// TwinCAT 3 PLC project Hexapod_Robot_Control_Test
// ProgramVersion: 3.1.4020.4
// libraries:
//   Tc2_MC2, * (Beckhoff Automation GmbH)
//   Tc2_Standard, * (Beckhoff Automation GmbH)
//   Tc2_System, * (Beckhoff Automation GmbH)
//   Tc3_Module, * (Beckhoff Automation GmbH)
//   VisuDialogs, * (System)
// project tree:
//   DUTs/Axis/ Axis.TcPOU (not stored)
//   DUTs/Delay/ Delay.TcPOU (not stored)
//   DUTs/Filter_Current/ E_TcMatSimDataAreaType_1.TcDUT (not stored), FB_Filter_Current_Hexapod_Robot.TcPOU (not stored), FB_TcMatSimObject_1.TcPOU (not stored), ST_Filter_Current_Hexapod_Robot_InitData.TcDUT (not stored), ST_Filter_Current_Hexapod_Robot_Input.TcDUT (not stored), ST_Filter_Current_Hexapod_Robot_Output.TcDUT (not stored), ST_TcMatSimObjectDataAreaInfo_1.TcDUT (not stored)
//   DUTs/Hexapod_Leg/ Hexapod_Leg.TcPOU (not stored)
//   DUTs/Mapping/ Hexapod_Robot_Mapping.TcPOU (not stored)
//   DUTs/Robot_Simulink/ E_TcMatSimDataAreaType.TcDUT, FB_HexMove.TcPOU, FB_TcMatSimObject.TcPOU (not stored), ST_HexMove_InitData.TcDUT (not stored), ST_HexMove_Input.TcDUT (not stored), ST_HexMove_Output.TcDUT, ST_TcMatSimObjectDataAreaInfo.TcDUT
//   / GlobalTextList.TcGTLO, PlcTask.TcTTO, 视图管理器.TcVMO (not stored)
//   POUs/ MAIN.TcPOU
//   VISUs/ Visu_Home.TcVIS (not stored), Visu_SimulinkMove.TcVIS, Visu_Power.TcVIS (not stored), Visu_Reset.TcVIS (not stored), Visu_Stand.TcVIS (not stored)
// real-time tasks:
//   TASK PlcTask: cycle T#1ms, priority 20, ADS port 350
// motion (NC):
//   TASK NC-Task 1 SAF: cycle T#1ms, priority 4, ADS port 501
//   TASK NC-Task 1 SVB: cycle T#1ms, priority 8, ADS port 511
//   AXIS Axis 1 (id 1)
//     Velo: SlowManual=10, FastManual=20
//     OtherSettings: AllowMotionCmdToSlave=true
//     encoder EncType=19
//       EncPara: ScaleFactorNumerator=0.000152590218967, MaxCount=#xffffffff
//     drive DrvType=16
//       DrvPara: MaxCount=#xffffffff
//         TimeComp: TaskDelayCycles=1
//     controller CtrType=1
//       CtrPara: PriorControlFactor=1
//         Observer: BandWidth=20
//   AXIS Axis 2 (id 2)
//     Velo: SlowManual=10, FastManual=20
//     OtherSettings: AllowMotionCmdToSlave=true
//     encoder EncType=19
//       EncPara: ScaleFactorNumerator=0.000152590218967, MaxCount=#xffffffff
//     drive DrvType=16
//       DrvPara: MaxCount=#xffffffff
//         TimeComp: TaskDelayCycles=1
//     controller CtrType=1
//       CtrPara: PriorControlFactor=1
//         Observer: BandWidth=20
//   AXIS Axis 3 (id 3)
//     Velo: SlowManual=10, FastManual=20
//     OtherSettings: AllowMotionCmdToSlave=true
//     encoder EncType=19
//       EncPara: ScaleFactorNumerator=0.000152590218967, MaxCount=#xffffffff
//     drive DrvType=16
//       DrvPara: MaxCount=#xffffffff
//         TimeComp: TaskDelayCycles=1
//     controller CtrType=1
//       CtrPara: PriorControlFactor=1
//         Observer: BandWidth=20
//   AXIS Axis 4 (id 4)
//     Velo: SlowManual=10, FastManual=20
//     OtherSettings: AllowMotionCmdToSlave=true
//     encoder EncType=19
//       EncPara: ScaleFactorNumerator=0.000152590218967, MaxCount=#xffffffff
//     drive DrvType=16
//       DrvPara: MaxCount=#xffffffff
//         TimeComp: TaskDelayCycles=1
//     controller CtrType=1
//       CtrPara: PriorControlFactor=1
//         Observer: BandWidth=20
//   AXIS Axis 5 (id 5)
//     Velo: SlowManual=10, FastManual=20
//     OtherSettings: AllowMotionCmdToSlave=true
//     encoder EncType=19
//       EncPara: ScaleFactorNumerator=0.000152590218967, MaxCount=#xffffffff
//     drive DrvType=16
//       DrvPara: MaxCount=#xffffffff
//         TimeComp: TaskDelayCycles=1
//     controller CtrType=1
//       CtrPara: PriorControlFactor=1
//         Observer: BandWidth=20
//   AXIS Axis 6 (id 6)
//     Velo: SlowManual=10, FastManual=20
//     OtherSettings: AllowMotionCmdToSlave=true
//     encoder EncType=19
//       EncPara: ScaleFactorNumerator=0.000152590218967, MaxCount=#xffffffff
//     drive DrvType=16
//       DrvPara: MaxCount=#xffffffff
//         TimeComp: TaskDelayCycles=1
//     controller CtrType=1
//       CtrPara: PriorControlFactor=1
//         Observer: BandWidth=20
//   AXIS Axis 7 (id 7)
//     Velo: SlowManual=10, FastManual=20
//     OtherSettings: AllowMotionCmdToSlave=true
//     encoder EncType=19
//       EncPara: ScaleFactorNumerator=0.000152590218967, MaxCount=#xffffffff
//     drive DrvType=16
//       DrvPara: MaxCount=#xffffffff
//         TimeComp: TaskDelayCycles=1
//     controller CtrType=1
//       CtrPara: PriorControlFactor=1
//         Observer: BandWidth=20
//   AXIS Axis 8 (id 8)
//     Velo: SlowManual=10, FastManual=20
//     OtherSettings: AllowMotionCmdToSlave=true
//     encoder EncType=19
//       EncPara: ScaleFactorNumerator=0.000152590218967, MaxCount=#xffffffff
//     drive DrvType=16
//       DrvPara: MaxCount=#xffffffff
//         TimeComp: TaskDelayCycles=1
//     controller CtrType=1
//       CtrPara: PriorControlFactor=1
//         Observer: BandWidth=20
//   AXIS Axis 9 (id 9)
//     Velo: SlowManual=10, FastManual=20
//     OtherSettings: AllowMotionCmdToSlave=true
//     encoder EncType=19
//       EncPara: ScaleFactorNumerator=0.000152590218967, MaxCount=#xffffffff
//     drive DrvType=16
//       DrvPara: MaxCount=#xffffffff
//         TimeComp: TaskDelayCycles=1
//     controller CtrType=1
//       CtrPara: PriorControlFactor=1
//         Observer: BandWidth=20
//   AXIS Axis 10 (id 10)
//     Velo: SlowManual=10, FastManual=20
//     OtherSettings: AllowMotionCmdToSlave=true
//     encoder EncType=19
//       EncPara: ScaleFactorNumerator=0.000152590218967, MaxCount=#xffffffff
//     drive DrvType=16
//       DrvPara: MaxCount=#xffffffff
//         TimeComp: TaskDelayCycles=1
//     controller CtrType=1
//       CtrPara: PriorControlFactor=1
//         Observer: BandWidth=20
//   AXIS Axis 11 (id 11)
//     Velo: SlowManual=10, FastManual=20
//     OtherSettings: AllowMotionCmdToSlave=true
//     encoder EncType=19
//       EncPara: ScaleFactorNumerator=0.000152590218967, MaxCount=#xffffffff
//     drive DrvType=16
//       DrvPara: MaxCount=#xffffffff
//         TimeComp: TaskDelayCycles=1
//     controller CtrType=1
//       CtrPara: PriorControlFactor=1
//         Observer: BandWidth=20
//   AXIS Axis 12 (id 12)
//     Velo: SlowManual=10, FastManual=20
//     OtherSettings: AllowMotionCmdToSlave=true
//     encoder EncType=19
//       EncPara: ScaleFactorNumerator=0.000152590218967, MaxCount=#xffffffff
//     drive DrvType=16
//       DrvPara: MaxCount=#xffffffff
//         TimeComp: TaskDelayCycles=1
//     controller CtrType=1
//       CtrPara: PriorControlFactor=1
//         Observer: BandWidth=20
//   AXIS Axis 13 (id 13)
//     Velo: SlowManual=10, FastManual=20
//     OtherSettings: AllowMotionCmdToSlave=true
//     encoder EncType=19
//       EncPara: ScaleFactorNumerator=0.000152590218967, MaxCount=#xffffffff
//     drive DrvType=16
//       DrvPara: MaxCount=#xffffffff
//         TimeComp: TaskDelayCycles=1
//     controller CtrType=1
//       CtrPara: PriorControlFactor=1
//         Observer: BandWidth=20
//   AXIS Axis 14 (id 14)
//     Velo: SlowManual=10, FastManual=20
//     OtherSettings: AllowMotionCmdToSlave=true
//     encoder EncType=19
//       EncPara: ScaleFactorNumerator=0.000152590218967, MaxCount=#xffffffff
//     drive DrvType=16
//       DrvPara: MaxCount=#xffffffff
//         TimeComp: TaskDelayCycles=1
//     controller CtrType=1
//       CtrPara: PriorControlFactor=1
//         Observer: BandWidth=20
//   AXIS Axis 15 (id 15)
//     Velo: SlowManual=10, FastManual=20
//     OtherSettings: AllowMotionCmdToSlave=true
//     encoder EncType=19
//       EncPara: ScaleFactorNumerator=0.000152590218967, MaxCount=#xffffffff
//     drive DrvType=16
//       DrvPara: MaxCount=#xffffffff
//         TimeComp: TaskDelayCycles=1
//     controller CtrType=1
//       CtrPara: PriorControlFactor=1
//         Observer: BandWidth=20
//   AXIS Axis 16 (id 16)
//     Velo: SlowManual=10, FastManual=20
//     OtherSettings: AllowMotionCmdToSlave=true
//     encoder EncType=19
//       EncPara: ScaleFactorNumerator=0.000152590218967, MaxCount=#xffffffff
//     drive DrvType=16
//       DrvPara: MaxCount=#xffffffff
//         TimeComp: TaskDelayCycles=1
//     controller CtrType=1
//       CtrPara: PriorControlFactor=1
//         Observer: BandWidth=20
//   AXIS Axis 17 (id 17)
//     Velo: SlowManual=10, FastManual=20
//     OtherSettings: AllowMotionCmdToSlave=true
//     encoder EncType=19
//       EncPara: ScaleFactorNumerator=0.000152590218967, MaxCount=#xffffffff
//     drive DrvType=16
//       DrvPara: MaxCount=#xffffffff
//         TimeComp: TaskDelayCycles=1
//     controller CtrType=1
//       CtrPara: PriorControlFactor=1
//         Observer: BandWidth=20
//   AXIS Axis 18 (id 18)
//     Velo: SlowManual=10, FastManual=20
//     OtherSettings: AllowMotionCmdToSlave=true
//     encoder EncType=19
//       EncPara: ScaleFactorNumerator=0.000152590218967, MaxCount=#xffffffff
//     drive DrvType=16
//       DrvPara: MaxCount=#xffffffff
//         TimeComp: TaskDelayCycles=1
//     controller CtrType=1
//       CtrPara: PriorControlFactor=1
//         Observer: BandWidth=20
// I/O:
//   DEVICE Device 3 (EtherCAT), AmsNetId 5.41.150.106.4.1
//     Drive 1 (Elmo Drive) [Gold EtherCAT GCON Drive Rev:0x000103F6]
//     Drive 2 (Elmo Drive) [Gold EtherCAT GCON Drive Rev:0x000103F6]
//     Drive 3 (Elmo Drive) [Gold EtherCAT GCON Drive Rev:0x000103F6]
//     Drive 4 (Elmo Drive) [Gold EtherCAT GCON Drive Rev:0x000103F6]
//     Drive 5 (Elmo Drive) [Gold EtherCAT GCON Drive Rev:0x000103F6]
//     Drive 6 (Elmo Drive) [Gold EtherCAT GCON Drive Rev:0x000103F6]
//     Drive 7 (Elmo Drive) [Gold EtherCAT GCON Drive Rev:0x000103F6]
//     Drive 8 (Elmo Drive) [Gold EtherCAT GCON Drive Rev:0x000103F6]
//     Drive 9 (Elmo Drive) [Gold EtherCAT GCON Drive Rev:0x000103F6]
//     Drive 10 (Elmo Drive) [Gold EtherCAT GCON Drive Rev:0x000103F6]
//     Drive 11 (Elmo Drive) [Gold EtherCAT GCON Drive Rev:0x000103F6]
//     Drive 12 (Elmo Drive) [Gold EtherCAT GCON Drive Rev:0x000103F6]
//     Drive 13 (Elmo Drive) [Gold EtherCAT GCON Drive Rev:0x000103F6]
//     Drive 14 (Elmo Drive) [Gold EtherCAT GCON Drive Rev:0x000103F6]
//     Drive 15 (Elmo Drive) [Gold EtherCAT GCON Drive Rev:0x000103F6]
//     Drive 16 (Elmo Drive) [Gold EtherCAT GCON Drive Rev:0x000103F6]
//     Drive 17 (Elmo Drive) [Gold EtherCAT GCON Drive Rev:0x000103F6]
//     Drive 18 (Elmo Drive) [Gold EtherCAT GCON Drive Rev:0x000103F6]
// variable links:
//   NC-Task 1 SAF/Axes/Axis 1 <-> Device 3 (EtherCAT)/Drive 1 (Elmo Drive)
//     Drive/Inputs/In/nDcOutputTime <-> InfoData/DcOutputShift
//     Drive/Inputs/In/nState1 <-> Inputs/Status word
//     Drive/Inputs/In/nState2 <-> Inputs/Status word @bit 8
//     Drive/Inputs/In/nState4 @bit 1 <-> WcState/InputToggle
//     Drive/Inputs/In/nState4 <-> WcState/WcState
//     Drive/Outputs/Out/nCtrl1 <-> Outputs/Control word
//     Drive/Outputs/Out/nCtrl2 <-> Outputs/Control word @bit 8
//     Drive/Outputs/Out/nDataOut1 <-> Outputs/Target Position
//     Enc/Inputs/In/nDataIn1 <-> Inputs/Position actual value
//     Enc/Inputs/In/nDcInputTime <-> InfoData/DcInputShift
//     Enc/Inputs/In/nState4 @bit 1 <-> WcState/InputToggle
//     Enc/Inputs/In/nState4 <-> WcState/WcState
//   NC-Task 1 SAF/Axes/Axis 10 <-> Device 3 (EtherCAT)/Drive 10 (Elmo Drive)
//     Drive/Inputs/In/nDcOutputTime <-> InfoData/DcOutputShift
//     Drive/Inputs/In/nState1 <-> Inputs/Status word
//     Drive/Inputs/In/nState2 <-> Inputs/Status word @bit 8
//     Drive/Inputs/In/nState4 @bit 1 <-> WcState/InputToggle
//     Drive/Inputs/In/nState4 <-> WcState/WcState
//     Drive/Outputs/Out/nCtrl1 <-> Outputs/Control word
//     Drive/Outputs/Out/nCtrl2 <-> Outputs/Control word @bit 8
//     Drive/Outputs/Out/nDataOut1 <-> Outputs/Target Position
//     Enc/Inputs/In/nDataIn1 <-> Inputs/Position actual value
//     Enc/Inputs/In/nDcInputTime <-> InfoData/DcInputShift
//     Enc/Inputs/In/nState4 @bit 1 <-> WcState/InputToggle
//     Enc/Inputs/In/nState4 <-> WcState/WcState
//   NC-Task 1 SAF/Axes/Axis 11 <-> Device 3 (EtherCAT)/Drive 11 (Elmo Drive)
//     Drive/Inputs/In/nDcOutputTime <-> InfoData/DcOutputShift
//     Drive/Inputs/In/nState1 <-> Inputs/Status word
//     Drive/Inputs/In/nState2 <-> Inputs/Status word @bit 8
//     Drive/Inputs/In/nState4 @bit 1 <-> WcState/InputToggle
//     Drive/Inputs/In/nState4 <-> WcState/WcState
//     Drive/Outputs/Out/nCtrl1 <-> Outputs/Control word
//     Drive/Outputs/Out/nCtrl2 <-> Outputs/Control word @bit 8
//     Drive/Outputs/Out/nDataOut1 <-> Outputs/Target Position
//     Enc/Inputs/In/nDataIn1 <-> Inputs/Position actual value
//     Enc/Inputs/In/nDcInputTime <-> InfoData/DcInputShift
//     Enc/Inputs/In/nState4 @bit 1 <-> WcState/InputToggle
//     Enc/Inputs/In/nState4 <-> WcState/WcState
//   NC-Task 1 SAF/Axes/Axis 12 <-> Device 3 (EtherCAT)/Drive 12 (Elmo Drive)
//     Drive/Inputs/In/nDcOutputTime <-> InfoData/DcOutputShift
//     Drive/Inputs/In/nState1 <-> Inputs/Status word
//     Drive/Inputs/In/nState2 <-> Inputs/Status word @bit 8
//     Drive/Inputs/In/nState4 @bit 1 <-> WcState/InputToggle
//     Drive/Inputs/In/nState4 <-> WcState/WcState
//     Drive/Outputs/Out/nCtrl1 <-> Outputs/Control word
//     Drive/Outputs/Out/nCtrl2 <-> Outputs/Control word @bit 8
//     Drive/Outputs/Out/nDataOut1 <-> Outputs/Target Position
//     Enc/Inputs/In/nDataIn1 <-> Inputs/Position actual value
//     Enc/Inputs/In/nDcInputTime <-> InfoData/DcInputShift
//     Enc/Inputs/In/nState4 @bit 1 <-> WcState/InputToggle
//     Enc/Inputs/In/nState4 <-> WcState/WcState
//   NC-Task 1 SAF/Axes/Axis 13 <-> Device 3 (EtherCAT)/Drive 13 (Elmo Drive)
//     Drive/Inputs/In/nDcOutputTime <-> InfoData/DcOutputShift
//     Drive/Inputs/In/nState1 <-> Inputs/Status word
//     Drive/Inputs/In/nState2 <-> Inputs/Status word @bit 8
//     Drive/Inputs/In/nState4 @bit 1 <-> WcState/InputToggle
//     Drive/Inputs/In/nState4 <-> WcState/WcState
//     Drive/Outputs/Out/nCtrl1 <-> Outputs/Control word
//     Drive/Outputs/Out/nCtrl2 <-> Outputs/Control word @bit 8
//     Drive/Outputs/Out/nDataOut1 <-> Outputs/Target Position
//     Enc/Inputs/In/nDataIn1 <-> Inputs/Position actual value
//     Enc/Inputs/In/nDcInputTime <-> InfoData/DcInputShift
//     Enc/Inputs/In/nState4 @bit 1 <-> WcState/InputToggle
//     Enc/Inputs/In/nState4 <-> WcState/WcState
//   NC-Task 1 SAF/Axes/Axis 14 <-> Device 3 (EtherCAT)/Drive 14 (Elmo Drive)
//     Drive/Inputs/In/nDcOutputTime <-> InfoData/DcOutputShift
//     Drive/Inputs/In/nState1 <-> Inputs/Status word
//     Drive/Inputs/In/nState2 <-> Inputs/Status word @bit 8
//     Drive/Inputs/In/nState4 @bit 1 <-> WcState/InputToggle
//     Drive/Inputs/In/nState4 <-> WcState/WcState
//     Drive/Outputs/Out/nCtrl1 <-> Outputs/Control word
//     Drive/Outputs/Out/nCtrl2 <-> Outputs/Control word @bit 8
//     Drive/Outputs/Out/nDataOut1 <-> Outputs/Target Position
//     Enc/Inputs/In/nDataIn1 <-> Inputs/Position actual value
//     Enc/Inputs/In/nDcInputTime <-> InfoData/DcInputShift
//     Enc/Inputs/In/nState4 @bit 1 <-> WcState/InputToggle
//     Enc/Inputs/In/nState4 <-> WcState/WcState
//   NC-Task 1 SAF/Axes/Axis 15 <-> Device 3 (EtherCAT)/Drive 15 (Elmo Drive)
//     Drive/Inputs/In/nDcOutputTime <-> InfoData/DcOutputShift
//     Drive/Inputs/In/nState1 <-> Inputs/Status word
//     Drive/Inputs/In/nState2 <-> Inputs/Status word @bit 8
//     Drive/Inputs/In/nState4 @bit 1 <-> WcState/InputToggle
//     Drive/Inputs/In/nState4 <-> WcState/WcState
//     Drive/Outputs/Out/nCtrl1 <-> Outputs/Control word
//     Drive/Outputs/Out/nCtrl2 <-> Outputs/Control word @bit 8
//     Drive/Outputs/Out/nDataOut1 <-> Outputs/Target Position
//     Enc/Inputs/In/nDataIn1 <-> Inputs/Position actual value
//     Enc/Inputs/In/nDcInputTime <-> InfoData/DcInputShift
//     Enc/Inputs/In/nState4 @bit 1 <-> WcState/InputToggle
//     Enc/Inputs/In/nState4 <-> WcState/WcState
//   NC-Task 1 SAF/Axes/Axis 16 <-> Device 3 (EtherCAT)/Drive 16 (Elmo Drive)
//     Drive/Inputs/In/nDcOutputTime <-> InfoData/DcOutputShift
//     Drive/Inputs/In/nState1 <-> Inputs/Status word
//     Drive/Inputs/In/nState2 <-> Inputs/Status word @bit 8
//     Drive/Inputs/In/nState4 @bit 1 <-> WcState/InputToggle
//     Drive/Inputs/In/nState4 <-> WcState/WcState
//     Drive/Outputs/Out/nCtrl1 <-> Outputs/Control word
//     Drive/Outputs/Out/nCtrl2 <-> Outputs/Control word @bit 8
//     Drive/Outputs/Out/nDataOut1 <-> Outputs/Target Position
//     Enc/Inputs/In/nDataIn1 <-> Inputs/Position actual value
//     Enc/Inputs/In/nDcInputTime <-> InfoData/DcInputShift
//     Enc/Inputs/In/nState4 @bit 1 <-> WcState/InputToggle
//     Enc/Inputs/In/nState4 <-> WcState/WcState
//   NC-Task 1 SAF/Axes/Axis 17 <-> Device 3 (EtherCAT)/Drive 17 (Elmo Drive)
//     Drive/Inputs/In/nDcOutputTime <-> InfoData/DcOutputShift
//     Drive/Inputs/In/nState1 <-> Inputs/Status word
//     Drive/Inputs/In/nState2 <-> Inputs/Status word @bit 8
//     Drive/Inputs/In/nState4 @bit 1 <-> WcState/InputToggle
//     Drive/Inputs/In/nState4 <-> WcState/WcState
//     Drive/Outputs/Out/nCtrl1 <-> Outputs/Control word
//     Drive/Outputs/Out/nCtrl2 <-> Outputs/Control word @bit 8
//     Drive/Outputs/Out/nDataOut1 <-> Outputs/Target Position
//     Enc/Inputs/In/nDataIn1 <-> Inputs/Position actual value
//     Enc/Inputs/In/nDcInputTime <-> InfoData/DcInputShift
//     Enc/Inputs/In/nState4 @bit 1 <-> WcState/InputToggle
//     Enc/Inputs/In/nState4 <-> WcState/WcState
//   NC-Task 1 SAF/Axes/Axis 18 <-> Device 3 (EtherCAT)/Drive 18 (Elmo Drive)
//     Drive/Inputs/In/nDcOutputTime <-> InfoData/DcOutputShift
//     Drive/Inputs/In/nState1 <-> Inputs/Status word
//     Drive/Inputs/In/nState2 <-> Inputs/Status word @bit 8
//     Drive/Inputs/In/nState4 @bit 1 <-> WcState/InputToggle
//     Drive/Inputs/In/nState4 <-> WcState/WcState
//     Drive/Outputs/Out/nCtrl1 <-> Outputs/Control word
//     Drive/Outputs/Out/nCtrl2 <-> Outputs/Control word @bit 8
//     Drive/Outputs/Out/nDataOut1 <-> Outputs/Target Position
//     Enc/Inputs/In/nDataIn1 <-> Inputs/Position actual value
//     Enc/Inputs/In/nDcInputTime <-> InfoData/DcInputShift
//     Enc/Inputs/In/nState4 @bit 1 <-> WcState/InputToggle
//     Enc/Inputs/In/nState4 <-> WcState/WcState
//   NC-Task 1 SAF/Axes/Axis 2 <-> Device 3 (EtherCAT)/Drive 2 (Elmo Drive)
//     Drive/Inputs/In/nDcOutputTime <-> InfoData/DcOutputShift
//     Drive/Inputs/In/nState1 <-> Inputs/Status word
//     Drive/Inputs/In/nState2 <-> Inputs/Status word @bit 8
//     Drive/Inputs/In/nState4 @bit 1 <-> WcState/InputToggle
//     Drive/Inputs/In/nState4 <-> WcState/WcState
//     Drive/Outputs/Out/nCtrl1 <-> Outputs/Control word
//     Drive/Outputs/Out/nCtrl2 <-> Outputs/Control word @bit 8
//     Drive/Outputs/Out/nDataOut1 <-> Outputs/Target Position
//     Enc/Inputs/In/nDataIn1 <-> Inputs/Position actual value
//     Enc/Inputs/In/nDcInputTime <-> InfoData/DcInputShift
//     Enc/Inputs/In/nState4 @bit 1 <-> WcState/InputToggle
//     Enc/Inputs/In/nState4 <-> WcState/WcState
//   NC-Task 1 SAF/Axes/Axis 3 <-> Device 3 (EtherCAT)/Drive 3 (Elmo Drive)
//     Drive/Inputs/In/nDcOutputTime <-> InfoData/DcOutputShift
//     Drive/Inputs/In/nState1 <-> Inputs/Status word
//     Drive/Inputs/In/nState2 <-> Inputs/Status word @bit 8
//     Drive/Inputs/In/nState4 @bit 1 <-> WcState/InputToggle
//     Drive/Inputs/In/nState4 <-> WcState/WcState
//     Drive/Outputs/Out/nCtrl1 <-> Outputs/Control word
//     Drive/Outputs/Out/nCtrl2 <-> Outputs/Control word @bit 8
//     Drive/Outputs/Out/nDataOut1 <-> Outputs/Target Position
//     Enc/Inputs/In/nDataIn1 <-> Inputs/Position actual value
//     Enc/Inputs/In/nDcInputTime <-> InfoData/DcInputShift
//     Enc/Inputs/In/nState4 @bit 1 <-> WcState/InputToggle
//     Enc/Inputs/In/nState4 <-> WcState/WcState
//   NC-Task 1 SAF/Axes/Axis 4 <-> Device 3 (EtherCAT)/Drive 4 (Elmo Drive)
//     Drive/Inputs/In/nDcOutputTime <-> InfoData/DcOutputShift
//     Drive/Inputs/In/nState1 <-> Inputs/Status word
//     Drive/Inputs/In/nState2 <-> Inputs/Status word @bit 8
//     Drive/Inputs/In/nState4 @bit 1 <-> WcState/InputToggle
//     Drive/Inputs/In/nState4 <-> WcState/WcState
//     Drive/Outputs/Out/nCtrl1 <-> Outputs/Control word
//     Drive/Outputs/Out/nCtrl2 <-> Outputs/Control word @bit 8
//     Drive/Outputs/Out/nDataOut1 <-> Outputs/Target Position
//     Enc/Inputs/In/nDataIn1 <-> Inputs/Position actual value
//     Enc/Inputs/In/nDcInputTime <-> InfoData/DcInputShift
//     Enc/Inputs/In/nState4 @bit 1 <-> WcState/InputToggle
//     Enc/Inputs/In/nState4 <-> WcState/WcState
//   NC-Task 1 SAF/Axes/Axis 5 <-> Device 3 (EtherCAT)/Drive 5 (Elmo Drive)
//     Drive/Inputs/In/nDcOutputTime <-> InfoData/DcOutputShift
//     Drive/Inputs/In/nState1 <-> Inputs/Status word
//     Drive/Inputs/In/nState2 <-> Inputs/Status word @bit 8
//     Drive/Inputs/In/nState4 @bit 1 <-> WcState/InputToggle
//     Drive/Inputs/In/nState4 <-> WcState/WcState
//     Drive/Outputs/Out/nCtrl1 <-> Outputs/Control word
//     Drive/Outputs/Out/nCtrl2 <-> Outputs/Control word @bit 8
//     Drive/Outputs/Out/nDataOut1 <-> Outputs/Target Position
//     Enc/Inputs/In/nDataIn1 <-> Inputs/Position actual value
//     Enc/Inputs/In/nDcInputTime <-> InfoData/DcInputShift
//     Enc/Inputs/In/nState4 @bit 1 <-> WcState/InputToggle
//     Enc/Inputs/In/nState4 <-> WcState/WcState
//   NC-Task 1 SAF/Axes/Axis 6 <-> Device 3 (EtherCAT)/Drive 6 (Elmo Drive)
//     Drive/Inputs/In/nDcOutputTime <-> InfoData/DcOutputShift
//     Drive/Inputs/In/nState1 <-> Inputs/Status word
//     Drive/Inputs/In/nState2 <-> Inputs/Status word @bit 8
//     Drive/Inputs/In/nState4 @bit 1 <-> WcState/InputToggle
//     Drive/Inputs/In/nState4 <-> WcState/WcState
//     Drive/Outputs/Out/nCtrl1 <-> Outputs/Control word
//     Drive/Outputs/Out/nCtrl2 <-> Outputs/Control word @bit 8
//     Drive/Outputs/Out/nDataOut1 <-> Outputs/Target Position
//     Enc/Inputs/In/nDataIn1 <-> Inputs/Position actual value
//     Enc/Inputs/In/nDcInputTime <-> InfoData/DcInputShift
//     Enc/Inputs/In/nState4 @bit 1 <-> WcState/InputToggle
//     Enc/Inputs/In/nState4 <-> WcState/WcState
//   NC-Task 1 SAF/Axes/Axis 7 <-> Device 3 (EtherCAT)/Drive 7 (Elmo Drive)
//     Drive/Inputs/In/nDcOutputTime <-> InfoData/DcOutputShift
//     Drive/Inputs/In/nState1 <-> Inputs/Status word
//     Drive/Inputs/In/nState2 <-> Inputs/Status word @bit 8
//     Drive/Inputs/In/nState4 @bit 1 <-> WcState/InputToggle
//     Drive/Inputs/In/nState4 <-> WcState/WcState
//     Drive/Outputs/Out/nCtrl1 <-> Outputs/Control word
//     Drive/Outputs/Out/nCtrl2 <-> Outputs/Control word @bit 8
//     Drive/Outputs/Out/nDataOut1 <-> Outputs/Target Position
//     Enc/Inputs/In/nDataIn1 <-> Inputs/Position actual value
//     Enc/Inputs/In/nDcInputTime <-> InfoData/DcInputShift
//     Enc/Inputs/In/nState4 @bit 1 <-> WcState/InputToggle
//     Enc/Inputs/In/nState4 <-> WcState/WcState
//   NC-Task 1 SAF/Axes/Axis 8 <-> Device 3 (EtherCAT)/Drive 8 (Elmo Drive)
//     Drive/Inputs/In/nDcOutputTime <-> InfoData/DcOutputShift
//     Drive/Inputs/In/nState1 <-> Inputs/Status word
//     Drive/Inputs/In/nState2 <-> Inputs/Status word @bit 8
//     Drive/Inputs/In/nState4 @bit 1 <-> WcState/InputToggle
//     Drive/Inputs/In/nState4 <-> WcState/WcState
//     Drive/Outputs/Out/nCtrl1 <-> Outputs/Control word
//     Drive/Outputs/Out/nCtrl2 <-> Outputs/Control word @bit 8
//     Drive/Outputs/Out/nDataOut1 <-> Outputs/Target Position
//     Enc/Inputs/In/nDataIn1 <-> Inputs/Position actual value
//     Enc/Inputs/In/nDcInputTime <-> InfoData/DcInputShift
//     Enc/Inputs/In/nState4 @bit 1 <-> WcState/InputToggle
//     Enc/Inputs/In/nState4 <-> WcState/WcState
//   NC-Task 1 SAF/Axes/Axis 9 <-> Device 3 (EtherCAT)/Drive 9 (Elmo Drive)
//     Drive/Inputs/In/nDcOutputTime <-> InfoData/DcOutputShift
//     Drive/Inputs/In/nState1 <-> Inputs/Status word
//     Drive/Inputs/In/nState2 <-> Inputs/Status word @bit 8
//     Drive/Inputs/In/nState4 @bit 1 <-> WcState/InputToggle
//     Drive/Inputs/In/nState4 <-> WcState/WcState
//     Drive/Outputs/Out/nCtrl1 <-> Outputs/Control word
//     Drive/Outputs/Out/nCtrl2 <-> Outputs/Control word @bit 8
//     Drive/Outputs/Out/nDataOut1 <-> Outputs/Target Position
//     Enc/Inputs/In/nDataIn1 <-> Inputs/Position actual value
//     Enc/Inputs/In/nDcInputTime <-> InfoData/DcInputShift
//     Enc/Inputs/In/nState4 @bit 1 <-> WcState/InputToggle
//     Enc/Inputs/In/nState4 <-> WcState/WcState
//   Hexapod_Robot_Control_Test/Hexapod_Robot_Control_Test Instance <-> Device 3 (EtherCAT)/Drive 1 (Elmo Drive)
//     PlcTask Inputs/MAIN.Current_Turque_Value[1] <-> Inputs_1/Current actual value
//   Hexapod_Robot_Control_Test/Hexapod_Robot_Control_Test Instance <-> Device 3 (EtherCAT)/Drive 10 (Elmo Drive)
//     PlcTask Inputs/MAIN.Current_Turque_Value[10] <-> Inputs_1/Current actual value
//   Hexapod_Robot_Control_Test/Hexapod_Robot_Control_Test Instance <-> Device 3 (EtherCAT)/Drive 11 (Elmo Drive)
//     PlcTask Inputs/MAIN.Current_Turque_Value[11] <-> Inputs_1/Current actual value
//   Hexapod_Robot_Control_Test/Hexapod_Robot_Control_Test Instance <-> Device 3 (EtherCAT)/Drive 12 (Elmo Drive)
//     PlcTask Inputs/MAIN.Current_Turque_Value[12] <-> Inputs_1/Current actual value
//   Hexapod_Robot_Control_Test/Hexapod_Robot_Control_Test Instance <-> Device 3 (EtherCAT)/Drive 13 (Elmo Drive)
//     PlcTask Inputs/MAIN.Current_Turque_Value[13] <-> Inputs_1/Current actual value
//   Hexapod_Robot_Control_Test/Hexapod_Robot_Control_Test Instance <-> Device 3 (EtherCAT)/Drive 14 (Elmo Drive)
//     PlcTask Inputs/MAIN.Current_Turque_Value[14] <-> Inputs_1/Current actual value
//   Hexapod_Robot_Control_Test/Hexapod_Robot_Control_Test Instance <-> Device 3 (EtherCAT)/Drive 15 (Elmo Drive)
//     PlcTask Inputs/MAIN.Current_Turque_Value[15] <-> Inputs_1/Current actual value
//   Hexapod_Robot_Control_Test/Hexapod_Robot_Control_Test Instance <-> Device 3 (EtherCAT)/Drive 16 (Elmo Drive)
//     PlcTask Inputs/MAIN.Current_Turque_Value[16] <-> Inputs_1/Current actual value
//   Hexapod_Robot_Control_Test/Hexapod_Robot_Control_Test Instance <-> Device 3 (EtherCAT)/Drive 17 (Elmo Drive)
//     PlcTask Inputs/MAIN.Current_Turque_Value[17] <-> Inputs_1/Current actual value
//   Hexapod_Robot_Control_Test/Hexapod_Robot_Control_Test Instance <-> Device 3 (EtherCAT)/Drive 18 (Elmo Drive)
//     PlcTask Inputs/MAIN.Current_Turque_Value[18] <-> Inputs_1/Current actual value
//   Hexapod_Robot_Control_Test/Hexapod_Robot_Control_Test Instance <-> Device 3 (EtherCAT)/Drive 2 (Elmo Drive)
//     PlcTask Inputs/MAIN.Current_Turque_Value[2] <-> Inputs_1/Current actual value
//   Hexapod_Robot_Control_Test/Hexapod_Robot_Control_Test Instance <-> Device 3 (EtherCAT)/Drive 3 (Elmo Drive)
//     PlcTask Inputs/MAIN.Current_Turque_Value[3] <-> Inputs_1/Current actual value
//   Hexapod_Robot_Control_Test/Hexapod_Robot_Control_Test Instance <-> Device 3 (EtherCAT)/Drive 4 (Elmo Drive)
//     PlcTask Inputs/MAIN.Current_Turque_Value[4] <-> Inputs_1/Current actual value
//   Hexapod_Robot_Control_Test/Hexapod_Robot_Control_Test Instance <-> Device 3 (EtherCAT)/Drive 5 (Elmo Drive)
//     PlcTask Inputs/MAIN.Current_Turque_Value[5] <-> Inputs_1/Current actual value
//   Hexapod_Robot_Control_Test/Hexapod_Robot_Control_Test Instance <-> Device 3 (EtherCAT)/Drive 6 (Elmo Drive)
//     PlcTask Inputs/MAIN.Current_Turque_Value[6] <-> Inputs_1/Current actual value
//   Hexapod_Robot_Control_Test/Hexapod_Robot_Control_Test Instance <-> Device 3 (EtherCAT)/Drive 7 (Elmo Drive)
//     PlcTask Inputs/MAIN.Current_Turque_Value[7] <-> Inputs_1/Current actual value
//   Hexapod_Robot_Control_Test/Hexapod_Robot_Control_Test Instance <-> Device 3 (EtherCAT)/Drive 8 (Elmo Drive)
//     PlcTask Inputs/MAIN.Current_Turque_Value[8] <-> Inputs_1/Current actual value
//   Hexapod_Robot_Control_Test/Hexapod_Robot_Control_Test Instance <-> Device 3 (EtherCAT)/Drive 9 (Elmo Drive)
//     PlcTask Inputs/MAIN.Current_Turque_Value[9] <-> Inputs_1/Current actual value
//   Hexapod_Robot_Control_Test/Hexapod_Robot_Control_Test Instance <-> NC-Task 1 SAF/Axes/Axis 1
//     PlcTask Inputs/MAIN.Axis_Robot[1].AxisRef.NcToPlc <-> Outputs/ToPlc
//     PlcTask Outputs/MAIN.Axis_Robot[1].AxisRef.PlcToNc <-> Inputs/FromPlc
//   Hexapod_Robot_Control_Test/Hexapod_Robot_Control_Test Instance <-> NC-Task 1 SAF/Axes/Axis 10
//     PlcTask Inputs/MAIN.Axis_Robot[10].AxisRef.NcToPlc <-> Outputs/ToPlc
//     PlcTask Outputs/MAIN.Axis_Robot[10].AxisRef.PlcToNc <-> Inputs/FromPlc
//   Hexapod_Robot_Control_Test/Hexapod_Robot_Control_Test Instance <-> NC-Task 1 SAF/Axes/Axis 11
//     PlcTask Inputs/MAIN.Axis_Robot[11].AxisRef.NcToPlc <-> Outputs/ToPlc
//     PlcTask Outputs/MAIN.Axis_Robot[11].AxisRef.PlcToNc <-> Inputs/FromPlc
//   Hexapod_Robot_Control_Test/Hexapod_Robot_Control_Test Instance <-> NC-Task 1 SAF/Axes/Axis 12
//     PlcTask Inputs/MAIN.Axis_Robot[12].AxisRef.NcToPlc <-> Outputs/ToPlc
//     PlcTask Outputs/MAIN.Axis_Robot[12].AxisRef.PlcToNc <-> Inputs/FromPlc
//   Hexapod_Robot_Control_Test/Hexapod_Robot_Control_Test Instance <-> NC-Task 1 SAF/Axes/Axis 13
//     PlcTask Inputs/MAIN.Axis_Robot[13].AxisRef.NcToPlc <-> Outputs/ToPlc
//     PlcTask Outputs/MAIN.Axis_Robot[13].AxisRef.PlcToNc <-> Inputs/FromPlc
//   Hexapod_Robot_Control_Test/Hexapod_Robot_Control_Test Instance <-> NC-Task 1 SAF/Axes/Axis 14
//     PlcTask Inputs/MAIN.Axis_Robot[14].AxisRef.NcToPlc <-> Outputs/ToPlc
//     PlcTask Outputs/MAIN.Axis_Robot[14].AxisRef.PlcToNc <-> Inputs/FromPlc
//   Hexapod_Robot_Control_Test/Hexapod_Robot_Control_Test Instance <-> NC-Task 1 SAF/Axes/Axis 15
//     PlcTask Inputs/MAIN.Axis_Robot[15].AxisRef.NcToPlc <-> Outputs/ToPlc
//     PlcTask Outputs/MAIN.Axis_Robot[15].AxisRef.PlcToNc <-> Inputs/FromPlc
//   Hexapod_Robot_Control_Test/Hexapod_Robot_Control_Test Instance <-> NC-Task 1 SAF/Axes/Axis 16
//     PlcTask Inputs/MAIN.Axis_Robot[16].AxisRef.NcToPlc <-> Outputs/ToPlc
//     PlcTask Outputs/MAIN.Axis_Robot[16].AxisRef.PlcToNc <-> Inputs/FromPlc
//   Hexapod_Robot_Control_Test/Hexapod_Robot_Control_Test Instance <-> NC-Task 1 SAF/Axes/Axis 17
//     PlcTask Inputs/MAIN.Axis_Robot[17].AxisRef.NcToPlc <-> Outputs/ToPlc
//     PlcTask Outputs/MAIN.Axis_Robot[17].AxisRef.PlcToNc <-> Inputs/FromPlc
//   Hexapod_Robot_Control_Test/Hexapod_Robot_Control_Test Instance <-> NC-Task 1 SAF/Axes/Axis 18
//     PlcTask Inputs/MAIN.Axis_Robot[18].AxisRef.NcToPlc <-> Outputs/ToPlc
//     PlcTask Outputs/MAIN.Axis_Robot[18].AxisRef.PlcToNc <-> Inputs/FromPlc
//   Hexapod_Robot_Control_Test/Hexapod_Robot_Control_Test Instance <-> NC-Task 1 SAF/Axes/Axis 2
//     PlcTask Inputs/MAIN.Axis_Robot[2].AxisRef.NcToPlc <-> Outputs/ToPlc
//     PlcTask Outputs/MAIN.Axis_Robot[2].AxisRef.PlcToNc <-> Inputs/FromPlc
//   Hexapod_Robot_Control_Test/Hexapod_Robot_Control_Test Instance <-> NC-Task 1 SAF/Axes/Axis 3
//     PlcTask Inputs/MAIN.Axis_Robot[3].AxisRef.NcToPlc <-> Outputs/ToPlc
//     PlcTask Outputs/MAIN.Axis_Robot[3].AxisRef.PlcToNc <-> Inputs/FromPlc
//   Hexapod_Robot_Control_Test/Hexapod_Robot_Control_Test Instance <-> NC-Task 1 SAF/Axes/Axis 4
//     PlcTask Inputs/MAIN.Axis_Robot[4].AxisRef.NcToPlc <-> Outputs/ToPlc
//     PlcTask Outputs/MAIN.Axis_Robot[4].AxisRef.PlcToNc <-> Inputs/FromPlc
//   Hexapod_Robot_Control_Test/Hexapod_Robot_Control_Test Instance <-> NC-Task 1 SAF/Axes/Axis 5
//     PlcTask Inputs/MAIN.Axis_Robot[5].AxisRef.NcToPlc <-> Outputs/ToPlc
//     PlcTask Outputs/MAIN.Axis_Robot[5].AxisRef.PlcToNc <-> Inputs/FromPlc
//   Hexapod_Robot_Control_Test/Hexapod_Robot_Control_Test Instance <-> NC-Task 1 SAF/Axes/Axis 6
//     PlcTask Inputs/MAIN.Axis_Robot[6].AxisRef.NcToPlc <-> Outputs/ToPlc
//     PlcTask Outputs/MAIN.Axis_Robot[6].AxisRef.PlcToNc <-> Inputs/FromPlc
//   Hexapod_Robot_Control_Test/Hexapod_Robot_Control_Test Instance <-> NC-Task 1 SAF/Axes/Axis 7
//     PlcTask Inputs/MAIN.Axis_Robot[7].AxisRef.NcToPlc <-> Outputs/ToPlc
//     PlcTask Outputs/MAIN.Axis_Robot[7].AxisRef.PlcToNc <-> Inputs/FromPlc
//   Hexapod_Robot_Control_Test/Hexapod_Robot_Control_Test Instance <-> NC-Task 1 SAF/Axes/Axis 8
//     PlcTask Inputs/MAIN.Axis_Robot[8].AxisRef.NcToPlc <-> Outputs/ToPlc
//     PlcTask Outputs/MAIN.Axis_Robot[8].AxisRef.PlcToNc <-> Inputs/FromPlc
//   Hexapod_Robot_Control_Test/Hexapod_Robot_Control_Test Instance <-> NC-Task 1 SAF/Axes/Axis 9
//     PlcTask Inputs/MAIN.Axis_Robot[9].AxisRef.NcToPlc <-> Outputs/ToPlc
//     PlcTask Outputs/MAIN.Axis_Robot[9].AxisRef.PlcToNc <-> Inputs/FromPlc

CONFIGURATION Hexapod_Robot_Control_Test
    RESOURCE PLC ON TwinCAT3
        TASK PlcTask(INTERVAL := T#1ms, PRIORITY := 20);
        PROGRAM MAIN WITH PlcTask : MAIN;
    END_RESOURCE
END_CONFIGURATION

// ---- DUTs/Robot_Simulink/E_TcMatSimDataAreaType.TcDUT
TYPE E_TcMatSimDataAreaType :
(
	NotSpecified := 0,
	Standard,
	InputSrc,
	InputDst,
	OutputSrc,
	OutputDst,
	InternalDa,
	MArea,
	RetainDa
);
END_TYPE

// ---- DUTs/Robot_Simulink/ST_HexMove_Output.TcDUT
TYPE ST_HexMove_Output :
STRUCT
	Disp_P: matrix_18_real_T;
END_STRUCT
END_TYPE

// ---- DUTs/Robot_Simulink/ST_TcMatSimObjectDataAreaInfo.TcDUT
TYPE ST_TcMatSimObjectDataAreaInfo :
STRUCT
	pPlcVar: PVOID;
	pModuleProcImg: PVOID;
	nSize: UDINT;
	nDataAreaId: UDINT;
	eDataAreaType: E_TcMatSimDataAreaType;
END_STRUCT
END_TYPE

// ---- POUs/MAIN.TcPOU

      PROGRAM MAIN
VAR
// =======================NC轴变量==========================
	//Leg_Robot			: ARRAY[1..6] OF Hexapod_Leg;	// 定义六足的腿
	Axis_Robot			: ARRAY[1..18] OF Axis;			// 定义六足轴参量(可以调整数据上限来调整电机数目)
	Axis_Delay			: Delay;						// 延迟程序
	Leg_Number			: INT;							// 定义机器人腿数
	Axis_Number 		: INT;							// 定义轴数目
	
	// ===================模块动作信号(按动作先后排列)==========
	Power_Execute 		: BOOL;							// 上电使能控制信号
	Axis_Power			: ARRAY[1..18] OF BOOL;			// 单电机使能
	Robot_Power			: BOOL;							// 机器人所有电机使能
	
	Home_Execute		: BOOL;							// 设置零点程序使能
	//Axis_Start_Back 	: ARRAY[1..18] OF BOOL;			// 单电机找零回退信号
	//Robot_Start_Back	: BOOL;							// 机器人所有电机回退信号
	Leg_Home_Set		: ARRAY[1..6] OF BOOL;	
	Axis_Home_Set		: ARRAY[1..18] OF BOOL;			// 单电机设定零点信号
	Robot_Home_Set		: BOOL;							// 机器人所有电机设定零点信号
	//Home_Set_Position	: ARRAY[1..18] OF LREAL;		// 找到零点后电机到达的位置
	//Delay_On			: ARRAY[1..18] OF BOOL;
	//TON1				: TON;
	
	Move_Execute		: BOOL;							// 绝对运动使能信号
	Robot_Stand_Execute	: BOOL;							// 机器人站立程序使能	
	Axis_Absolute_Eable	: ARRAY[1..18] OF BOOL;			// 单电机绝对运动使能信号
	Robot_Absolute_Eable: ARRAY[1..18] OF BOOL;			// 机器人站立使能信号
	Axis_Move_Position	: ARRAY[1..18] OF LREAL;		// 电机绝对运动位置			
	
	ExSetPoint_Execute	: BOOL;							// 机器人外部信号发生使能
	ExtSetPointEnable	: BOOL;							// 外部信号发生信号
	ExtSetPointDisable	: BOOL;							// 外部信号结束信号
	
	Reset_Execute		: BOOL;							// 电机驱动重置动作发生使能
	Axis_Reset			: ARRAY[1..18] OF BOOL;			// 单电机驱动重置信号使能
	Robot_Reset			: BOOL;							// 机器人整体电机驱动重置
	Axis_ResetDone		: ARRAY[1..18] OF BOOL;			// 单电机驱动重置完成
	
	// ===================状态监测变量=======================
	Power_Status	: ARRAY[1..18] OF BOOL;				// 上电监测信号
	Leg_Home_Done	: ARRAY[1..6] OF BOOL;
	Home_Done		: ARRAY[1..18] OF BOOL;				// 找零监测信号
	MoveAbsoluteDone: ARRAY[1..18] OF BOOL;				// 电机运动监测信号
	
	Robot_Error		: BOOL;								// 机器人电机错误信号
	Axis_Error		: ARRAY[1..18] OF BOOL;				// 电机错误监测信号
	Axis_ErrorID	: ARRAY[1..18] OF UDINT;			// 电机错误号码监测信号
	
	Axis_ActPostion	: ARRAY[1..18] OF LREAL;			// 电机轴实际位置
	Difference_Position	: ARRAY[1..18] OF LREAL;		// 实际位置与输入位置差值
	
	// =======================模块中间变量======================
	//HomeDone_Number	: LREAL :=0;					//完成找零的轴数
	//ExSetPoint_Position	: ARRAY[1..18] OF LREAL;		// 外部信号位置
	//t					: LREAL :=0;
	
	// =======================驱动器信号监测====================
	Current_Turque_Value  AT%IW0 : ARRAY[1..18] OF INT ;	//电流、力矩相关值
	Max_Turque_Value 	: INT ;							// 设置最大力矩边界值
	
		// ====================Simulink模块相关=====================
	Robot_Simulink		: FB_HexMove(oid:=16#01010020);	// Simulink模型定义
	Model_Position		: ARRAY[1..18] OF LREAL;			// Simulink中各个腿的位置
	ExSetPoint_Position	: ARRAY[1..18] OF LREAL;			// 外部信号位置
	T_ALL				: LREAL:=100;						// Simulink模型运动总时长
	t_Interval			: LREAL:=0.001;						// 取样时间间隔，默认为1ms
	t					: LREAL:=0;							// 取样当前时间变量，以0为起点
	Mapping				: Hexapod_Robot_Mapping;			// 变量映射			
	Home_Position 		: ARRAY[1..18] OF LREAL;			// Home结束后的位移值
  
  Filter_Current  : FB_Filter_Current_Hexapod_Robot(oid:=16#01010030);
  Current_Turque_Filter  : ARRAY[1..18] OF LREAL;
END_VAR

// =======================子程序使能(永久运行)===================
Variable_Monitor();			// 变量监测子程序使能
Logic_Control();			// 逻辑控制子程序使能
Variable_Set();				// 各动作速度子程序使能
SetGenerator();				// 外部信号发生子程序使能
Leg_Action();				// 单腿运动子程序使能
Robot_Action();				// 机器人整体运动子程序使能

// =====================电机驱动重置=============================
IF Reset_Execute THEN
	FOR Axis_Number := 1 TO 18 {BY 1} DO
		Axis_Robot[Axis_Number].Reset(Drive_Reset:= Axis_Reset[Axis_Number]);
	END_FOR
END_IF

// =======================电机上电===============================
IF Power_Execute THEN
	Filter_Current.Execute();
	FOR Axis_Number := 1 TO 18 {BY 1} DO
		Axis_Robot[Axis_Number].Power(Axis_Enable:= Axis_Power[Axis_Number]);
	END_FOR
END_IF

// =======================找零程序===============================
IF Home_Execute THEN
	Robot_Simulink.Execute();	// Simulink模型使能，用来为找零后的电机提供初始位移
	FOR Axis_Number := 1 TO 18 {BY 1} DO
		Axis_Robot[Axis_Number].Home(Drive_Home:= Axis_Home_Set[Axis_Number]);
	END_FOR
END_IF

// =======================站立程序===============================
IF Move_Execute THEN
	FOR Axis_Number := 1 TO 18 {BY 1} DO
		Axis_Robot[Axis_Number].Move_Absolute(	Drive_Move_Absolute:= Axis_Absolute_Eable[Axis_Number], 
												Absolute_Position:= Axis_Move_Position[Axis_Number]);
	END_FOR
END_IF
	
// =======================外部信号运动程序=======================
IF ExSetPoint_Execute THEN
	//SetGenerator();			// 使能外部信号发生子程序
	Robot_Simulink.Execute();	// Simulink模型使能
	FOR Axis_Number := 1 TO 18 {BY 1} DO
		Axis_Robot[Axis_Number].ExtSetPoint(Drive_ExtSetPointEnable:= ExtSetPointEnable, 
											Drive_ExtSetPointDisable:= ExtSetPointDisable, 
											ExSetPosition:= ExSetPoint_Position[Axis_Number]);
	END_FOR
END_IF

ACTION Leg_Action:
// ===================机器人单挑腿找零程序====================
IF Home_Execute THEN
	FOR Leg_Number := 1 TO 6 {BY 1} DO
		IF Leg_Home_Set[Leg_Number] THEN		// 在可视化中，Leg_Home_Set为点动
			Axis_Home_Set[1+(Leg_Number-1)*3] := Leg_Home_Set[Leg_Number];
			Axis_Home_Set[2+(Leg_Number-1)*3] := Leg_Home_Set[Leg_Number];
			Axis_Home_Set[3+(Leg_Number-1)*3] := Leg_Home_Set[Leg_Number];
		ELSIF Home_Done[1+(Leg_Number-1)*3] AND Axis_Home_Set[2+(Leg_Number-1)*3] AND Axis_Home_Set[3+(Leg_Number-1)*3] THEN
			Leg_Home_Set[Leg_Number] := FALSE; 
		END_IF
	END_FOR
END_IF
END_ACTION

ACTION Logic_Control:
// =======================控制逻辑区==========================
// 保证所有的动作拥有合理的先后顺序，优化控制逻辑
// 也防止出现两个或两个以上动作同时进行的情况，保证控制安全

// ===================电机驱动重置逻辑========================
//FOR Axis_Number := 1 TO 18 {BY 1} DO
IF Axis_Error[1] OR Axis_Error[2] OR Axis_Error[3] OR Axis_Error[4] OR Axis_Error[5] OR Axis_Error[6]
	 OR Axis_Error[7] OR Axis_Error[8] OR Axis_Error[9] OR Axis_Error[10] OR Axis_Error[11] OR Axis_Error[12]
		OR Axis_Error[13] OR Axis_Error[14] OR Axis_Error[15] OR Axis_Error[16] OR Axis_Error[17] OR Axis_Error[18]
THEN
	Robot_Error := TRUE;
ELSE
	Robot_Error := FALSE;
END_IF
//END_FOR

IF Robot_Error THEN
	Reset_Execute := TRUE;
ELSIF NOT Robot_Error THEN
	Reset_Execute := FALSE;
ELSIF NOT Reset_Execute THEN
	Axis_Reset[Axis_Number] := FALSE;
	Axis_Robot[Axis_Number].Reset(Drive_Reset:= Axis_Reset[Axis_Number]);
END_IF

// =====================上电程序逻辑==========================
IF NOT Power_Execute THEN
	FOR Axis_Number := 1 TO 18 {BY 1} DO
		Axis_Power[Axis_Number] := FALSE;
		Axis_Robot[Axis_Number].Power(Axis_Enable:= Axis_Power[Axis_Number]);
	END_FOR
END_IF

// =====================找零程序逻辑==========================
IF Home_Execute THEN
	FOR Axis_Number := 1 TO 18 {BY 1} DO
		IF Home_Done[Axis_Number] THEN			// 	丝杠到达零点位置后，单电j机标零使能位关闭			
			Axis_Home_Set[Axis_Number] :=0;	
			Axis_Robot[Axis_Number].Home(Drive_Home:= Axis_Home_Set[Axis_Number]);
		END_IF
	END_FOR
	Move_Execute :=0;							// 设定零点时，不能进行其他运动
	ExSetPoint_Execute :=0;
ELSIF NOT Home_Execute THEN
	FOR Axis_Number := 1 TO 18 {BY 1} DO
		//Axis_Start_Back[Axis_Number] :=0;
		Axis_Home_Set[Axis_Number] := 0;
	END_FOR
END_IF

// =====================机器人站立逻辑==========================
IF Move_Execute THEN
	//Absolute_Eable := TRUE;
	Home_Execute := FALSE;						// 站立运动使能时，机器人调零必须结束
	ExSetPoint_Execute :=0;						// 站立运动时，不能进行其他运动
	FOR Axis_Number := 1 TO 18 {BY 1} DO
		IF MoveAbsoluteDone[Axis_Number] THEN	// 	丝杠到达设定位置后，单电机绝对运动使能位关闭
			Axis_Absolute_Eable[Axis_Number] := FALSE;
		END_IF
	END_FOR
ELSIF NOT Move_Execute THEN						// 站立运动不使能,轴不能运动
	FOR Axis_Number := 1 TO 18 {BY 1} DO
		Axis_Absolute_Eable[Axis_Number] := FALSE;
		Axis_Robot[Axis_Number].Move_Absolute(	Drive_Move_Absolute:= Axis_Absolute_Eable[Axis_Number], 
												Absolute_Position:= Axis_Move_Position[Axis_Number]);
	END_FOR
END_IF

// =====================外部信号发生逻辑========================
IF ExSetPoint_Execute THEN
	Home_Execute := FALSE;						// 外部信号发生使能时，机器人调零必须结束
	Move_Execute :=0;							// 外部信号发生时，不能进行其他运动
ELSIF NOT ExSetPoint_Execute THEN
	ExtSetPointEnable := 0;						// 外部信号发生不使能时，外部信号不能进入程序
	ExtSetPointDisable :=0;
ELSIF ExtSetPointDisable THEN
	ExtSetPointEnable :=0;						// 外部信号发生停止与外部信号发生开始不能同时进行
END_IF
END_ACTION

ACTION Robot_Action:
// =================机器人整体运动命令区======================
// 六足所有电机整体控制

// ====================机器人驱动重置=========================
IF Robot_Reset THEN
	IF Reset_Execute THEN
		Axis_Reset[Axis_Number] := TRUE;
		FOR Axis_Number := 1 TO 18 {BY 1} DO
			Axis_Robot[Axis_Number].Reset(Drive_Reset:= Axis_Reset[Axis_Number]);
		END_FOR
	END_IF
END_IF	

// ===================机器人所有电机上电======================
IF Robot_Power THEN	
	IF Power_Execute THEN
		FOR Axis_Number := 1 TO 18 {BY 1} DO
			Axis_Power[Axis_Number] := TRUE ;
		END_FOR
	END_IF
END_IF
	
// ===================机器人找零程序=======================
IF Robot_Home_Set THEN				// 标零程序
	//Robot_Start_Back := FALSE;
	IF Home_Execute THEN
		Leg_Home_Set[3] := Leg_Home_Set[5] := Leg_Home_Set[1];	// 在整机调零时，1\3\5三条腿同时调零；
		Leg_Home_Set[4] := Leg_Home_Set[6] := Leg_Home_Set[2];	// 在整机调零时，2\4\6三条腿同时调零；
	ELSIF NOT Home_Execute THEN
		FOR Leg_Number := 1 TO 6 {BY 1} DO
			Leg_Home_Set[Leg_Number] := FALSE;
		END_FOR
	END_IF
ELSIF NOT Robot_Home_Set AND NOT Home_Execute THEN
	FOR Axis_Number := 1 TO 18 {BY 1} DO
	Axis_Home_Set[Axis_Number] := FALSE;
	END_FOR
END_IF

// =====================站立程序===============================
IF Robot_Stand_Execute THEN
	IF Move_Execute THEN
		FOR Axis_Number := 1 TO 18 {BY 1} DO
			IF MoveAbsoluteDone[Axis_Number] THEN		// 	丝杠到达设定位置后，单电机绝对运动使能位关闭
				Axis_Absolute_Eable[Axis_Number] := FALSE;
			ELSE
				Axis_Absolute_Eable[Axis_Number] := TRUE;
			END_IF
		END_FOR
	END_IF
ELSIF NOT Robot_Stand_Execute AND NOT Move_Execute THEN 
	FOR Axis_Number := 1 TO 18 {BY 1} DO
		Axis_Absolute_Eable[Axis_Number] := FALSE;
	END_FOR
END_IF

// ======================外部信号发生=========================
IF ExtSetPointEnable THEN	
	//FOR Axis_Number := 1 TO 2 {BY 1} DO
	t := t + t_Interval;
	ExtSetPointDisable := FALSE;
	//END_FOR
END_IF

IF t=0 THEN
	FOR Axis_Number := 1 TO 18 {BY 1} DO
		Home_Position[Axis_Number] := Axis_ActPostion[Axis_Number];
	END_FOR
ELSIF t>=T_ALL THEN
	ExtSetPointEnable := FALSE;
	t:=0;
	ExtSetPointDisable := TRUE;
END_IF
END_ACTION

ACTION SetGenerator:
// ====================外部信号发生测试区=====================
// 用来测试外部信号发生功能和电机相关参数

// =================外部信号正弦信号发生======================
(*IF ExtSetPointEnable THEN
	FOR Axis_Number := 1 TO 18 {BY 1} DO
		ExSetPoint_Position[Axis_Number]:=10*SIN(2*3.14*t);
		t := t+0.001;
	END_FOR
END_IF

// =================外部信号停止逻辑判断=======================
//IF Axis_Robot[Axis_Number].State_ExtSetPiontDone THEN
IF t>=20 THEN
	ExtSetPointEnable := FALSE;
	t:=0;
	ExtSetPointDisable := TRUE;
END_IF
//END_IF*)
END_ACTION

ACTION Variable_Monitor:
// =====================关键数据信号监测======================

// ==============最大力矩设置区(边界控制条件)=================
FOR Axis_Number := 1 TO 18 {BY 1} DO
	Axis_Robot[Axis_Number].Max_Turque_Value := Max_Turque_Value;
END_FOR

// =======================力矩检测区==========================
FOR Axis_Number := 1 TO 18 {BY 1} DO
	Axis_Robot[Axis_Number].Current_Turque_Value := Current_Turque_Value[Axis_Number];
END_FOR

// ====================轴实际位置检测区=======================
FOR Axis_Number := 1 TO 18 {BY 1} DO
	Axis_ActPostion[Axis_Number] := Axis_Robot[Axis_Number].ActPosition;
END_FOR

// =======================上电状态检测区======================
FOR Axis_Number := 1 TO 18 {BY 1} DO
	Power_Status[Axis_Number] := Axis_Robot[Axis_Number].State_PowerStatus;
END_FOR

// =======================找零状态检测区======================
FOR Axis_Number := 1 TO 18 {BY 1} DO
	Home_Done[Axis_Number] := Axis_Robot[Axis_Number].State_HomeDone;
END_FOR

(*FOR Leg_Number := 1 TO 6 {BY 1} DO
	Leg_Home_Done[Leg_Number] := Leg_Robot[Axis_Number].State_HomeDone;
END_FOR*)

// ===================电机绝对运动状态检测区==================
FOR Axis_Number := 1 TO 18 {BY 1} DO
	MoveAbsoluteDone[Axis_Number] := Axis_Robot[Axis_Number].State_MoveAbsoluteDone;
END_FOR

// =======================电机错误检测区======================
FOR Axis_Number := 1 TO 18 {BY 1} DO
	Axis_Error[Axis_Number] := Axis_Robot[Axis_Number].Axis_Error;
	Axis_ErrorID[Axis_Number] := Axis_Robot[Axis_Number].Axis_ErrorID;
END_FOR

// ==============实际运动位移和输入位移差值检测区==============
FOR Axis_Number := 1 TO 18 {BY 1} DO
	Difference_Position[Axis_Number] := Axis_ActPostion[Axis_Number]- Mapping.Controller_Leg_Position[Axis_Number]; 
END_FOR
END_ACTION

ACTION Variable_Set:
// =======================速度规定区==========================
FOR Axis_Number := 1 TO 18 {BY 1} DO						//此时每一个电机的速度都是一样的
	Axis_Robot[Axis_Number].Home_Velocity 	:= 20;			//找零速度(Axis_Jog中的速度)
	Axis_Robot[Axis_Number].Move_Relative_Velocity	:=30;	//相对运动速度
END_FOR
IF Home_Execute THEN
	//IF Robot_Home_Set THEN
		Axis_Robot[1].Move_Absolute_Velocity :=17; Axis_Robot[3].Move_Absolute_Velocity :=17; Axis_Robot[4].Move_Absolute_Velocity :=16.74;
		Axis_Robot[6].Move_Absolute_Velocity :=16.74; Axis_Robot[7].Move_Absolute_Velocity :=17.3; Axis_Robot[9].Move_Absolute_Velocity :=17.3;
		Axis_Robot[10].Move_Absolute_Velocity :=16.95; Axis_Robot[12].Move_Absolute_Velocity :=16.95; Axis_Robot[13].Move_Absolute_Velocity :=17;
		Axis_Robot[15].Move_Absolute_Velocity :=17; Axis_Robot[16].Move_Absolute_Velocity :=17; Axis_Robot[18].Move_Absolute_Velocity :=17;
		Axis_Robot[2].Move_Absolute_Velocity :=20; Axis_Robot[5].Move_Absolute_Velocity :=20; Axis_Robot[8].Move_Absolute_Velocity :=20;
		Axis_Robot[11].Move_Absolute_Velocity :=20; Axis_Robot[14].Move_Absolute_Velocity :=20; Axis_Robot[17].Move_Absolute_Velocity :=20;
	//ELSIF NOT Robot_Home_Set THEN
		//FOR Axis_Number := 1 TO 18 {BY 1} DO
			//Axis_Robot[Axis_Number].Move_Absolute_Velocity	:=10;
		//END_FOR
	//END_IF
ELSE
	FOR Axis_Number := 1 TO 18 {BY 1} DO
			Axis_Robot[Axis_Number].Move_Absolute_Velocity	:=10;
	END_FOR
END_IF
	

// =======================位置规定区==========================
FOR Axis_Number := 1 TO 18 {BY 1} DO
	Axis_Move_Position[Axis_Number] := 160;
END_FOR

// =====================最大力矩规定区========================
Max_Turque_Value := 1300;

// ===============电机设置零点后到达位置规定区================
(*Axis_Robot[1].Home_Absolute_Position := 73.7632; Axis_Robot[3].Home_Absolute_Position := 73.7632; Axis_Robot[4].Home_Absolute_Position := 73.7632;
Axis_Robot[6].Home_Absolute_Position := 73.7632; Axis_Robot[7].Home_Absolute_Position := 73.7632; Axis_Robot[9].Home_Absolute_Position := 73.7632;
Axis_Robot[10].Home_Absolute_Position := 73.7632; Axis_Robot[12].Home_Absolute_Position := 73.7632; Axis_Robot[13].Home_Absolute_Position := 73.7632;
Axis_Robot[15].Home_Absolute_Position := 73.7632; Axis_Robot[16].Home_Absolute_Position := 73.7632; Axis_Robot[18].Home_Absolute_Position := 73.7632;
Axis_Robot[2].Home_Absolute_Position := 83.7506; Axis_Robot[5].Home_Absolute_Position := 83.7506; Axis_Robot[8].Home_Absolute_Position := 83.7506;
Axis_Robot[11].Home_Absolute_Position := 83.7506; Axis_Robot[14].Home_Absolute_Position := 83.7506; Axis_Robot[17].Home_Absolute_Position := 83.7506;*)
(*Axis_Robot[1].Home_Absolute_Position := 138; Axis_Robot[3].Home_Absolute_Position := 138; Axis_Robot[4].Home_Absolute_Position := 138;
Axis_Robot[6].Home_Absolute_Position := 138; Axis_Robot[7].Home_Absolute_Position := 138; Axis_Robot[9].Home_Absolute_Position := 138;
Axis_Robot[10].Home_Absolute_Position := 138; Axis_Robot[12].Home_Absolute_Position := 138; Axis_Robot[13].Home_Absolute_Position := 138;
Axis_Robot[15].Home_Absolute_Position := 138; Axis_Robot[16].Home_Absolute_Position := 138; Axis_Robot[18].Home_Absolute_Position := 138;
Axis_Robot[2].Home_Absolute_Position := 149; Axis_Robot[5].Home_Absolute_Position := 149; Axis_Robot[8].Home_Absolute_Position := 149;
Axis_Robot[11].Home_Absolute_Position := 149; Axis_Robot[14].Home_Absolute_Position := 149; Axis_Robot[17].Home_Absolute_Position := 149;*)
FOR Axis_Number := 1 TO 18 {BY 1} DO
	Axis_Robot[Axis_Number].Home_Absolute_Position := Mapping.Controller_Leg_Position[Axis_Number];
END_FOR

// ===================外部信号发生电机位置输入值================
FOR Axis_Number := 1 TO 18 {BY 1} DO
	ExSetPoint_Position[Axis_Number]:= Mapping.Controller_Leg_Position[Axis_Number];
END_FOR

// ===================电机和腿映射关系========================
//FOR Leg_Number := 1 TO 6 {BY 1} DO
(*Leg_Robot[1](Axis1:= Axis_Robot[1], Axis2:= Axis_Robot[2], Axis3:= Axis_Robot[3]);
Leg_Robot[2](Axis1:= Axis_Robot[4], Axis2:= Axis_Robot[5], Axis3:= Axis_Robot[6]);
Leg_Robot[3](Axis1:= Axis_Robot[7], Axis2:= Axis_Robot[8], Axis3:= Axis_Robot[9]);
Leg_Robot[4](Axis1:= Axis_Robot[10], Axis2:= Axis_Robot[11], Axis3:= Axis_Robot[12]);
Leg_Robot[5](Axis1:= Axis_Robot[13], Axis2:= Axis_Robot[14], Axis3:= Axis_Robot[15]);
Leg_Robot[6](Axis1:= Axis_Robot[16], Axis2:= Axis_Robot[17], Axis3:= Axis_Robot[18]);*)
//END_FOR

// ===================程序与模型的变量链接===================
Mapping(Model_Leg_Position:= Model_Position);				// 映射运动学模型中腿编号和控制模型中的电机编号
Robot_Simulink.stInput.t := t;								// 采样时间t与Simulink模型中的采样时间链接
Model_Position := Robot_Simulink.stOutput.Disp_P;			// Simulink中的电机输出位移输入到控制模型
FOR Axis_Number := 1 TO 18 {BY 1} DO
	Filter_Current.stInput.Current_Motor[Axis_Number-1] := Current_Turque_Value[Axis_Number];
END_FOR	
Current_Turque_Filter := Filter_Current.stOutput.Current_Monitor;
END_ACTION

END_PROGRAM

// ---- DUTs/Robot_Simulink/FB_HexMove.TcPOU
{attribute 'TcDependOnClassFactory' := 'HexMove'}
FUNCTION_BLOCK FB_HexMove EXTENDS FB_TcMatSimObject
VAR_INPUT
	stInput: ST_HexMove_Input;
END_VAR
VAR_OUTPUT
	stOutput: ST_HexMove_Output;
END_VAR
VAR
	stInitData: ST_HexMove_InitData;
	arrDataAreas: ARRAY[1..2] OF ST_TcMatSimObjectDataAreaInfo;
	bParametersVerified: BOOL;
END_VAR

PROPERTY CallBy_Online : TctModuleCallByType
GET
hResult := GetObjPara(16#00000000,sizeof(CallBy_Online),adr(CallBy_Online));
END_GET
SET
hResult := SetObjPara(16#00000000,sizeof(CallBy_Online),adr(CallBy_Online));
END_SET
END_PROPERTY

PROPERTY CallBy_Startup : TctModuleCallByType
GET
CallBy_Startup := stInitData.CallBy;
END_GET
SET
stInitData.CallBy := CallBy_Startup;
END_SET
END_PROPERTY

PROPERTY ContextInfoArr_0_TaskCycleTimeNs_Online : UDINT
GET
hResult := GetObjPara(16#03002080,sizeof(ContextInfoArr_0_TaskCycleTimeNs_Online),adr(ContextInfoArr_0_TaskCycleTimeNs_Online));
END_GET
SET
hResult := SetObjPara(16#03002080,sizeof(ContextInfoArr_0_TaskCycleTimeNs_Online),adr(ContextInfoArr_0_TaskCycleTimeNs_Online));
END_SET
END_PROPERTY

PROPERTY ContextInfoArr_0_TaskCycleTimeNs_Startup : UDINT
GET
ContextInfoArr_0_TaskCycleTimeNs_Startup := stInitData.ContextInfoArr_0_TaskCycleTimeNs;
END_GET
SET
stInitData.ContextInfoArr_0_TaskCycleTimeNs := ContextInfoArr_0_TaskCycleTimeNs_Startup;
END_SET
END_PROPERTY

PROPERTY ContextInfoArr_0_TaskOid_Online : OTCID
GET
hResult := GetObjPara(16#03002060,sizeof(ContextInfoArr_0_TaskOid_Online),adr(ContextInfoArr_0_TaskOid_Online));
END_GET
SET
hResult := SetObjPara(16#03002060,sizeof(ContextInfoArr_0_TaskOid_Online),adr(ContextInfoArr_0_TaskOid_Online));
END_SET
END_PROPERTY

PROPERTY ContextInfoArr_0_TaskOid_Startup : OTCID
GET
ContextInfoArr_0_TaskOid_Startup := stInitData.ContextInfoArr_0_TaskOid;
END_GET
SET
stInitData.ContextInfoArr_0_TaskOid := ContextInfoArr_0_TaskOid_Startup;
END_SET
END_PROPERTY

PROPERTY ContextInfoArr_0_TaskPort_Online : UINT
GET
hResult := GetObjPara(16#03002090,sizeof(ContextInfoArr_0_TaskPort_Online),adr(ContextInfoArr_0_TaskPort_Online));
END_GET
SET
hResult := SetObjPara(16#03002090,sizeof(ContextInfoArr_0_TaskPort_Online),adr(ContextInfoArr_0_TaskPort_Online));
END_SET
END_PROPERTY

PROPERTY ContextInfoArr_0_TaskPort_Startup : UINT
GET
ContextInfoArr_0_TaskPort_Startup := stInitData.ContextInfoArr_0_TaskPort;
END_GET
SET
stInitData.ContextInfoArr_0_TaskPort := ContextInfoArr_0_TaskPort_Startup;
END_SET
END_PROPERTY

PROPERTY ContextInfoArr_0_TaskPriority_Online : UDINT
GET
hResult := GetObjPara(16#03002070,sizeof(ContextInfoArr_0_TaskPriority_Online),adr(ContextInfoArr_0_TaskPriority_Online));
END_GET
SET
hResult := SetObjPara(16#03002070,sizeof(ContextInfoArr_0_TaskPriority_Online),adr(ContextInfoArr_0_TaskPriority_Online));
END_SET
END_PROPERTY

PROPERTY ContextInfoArr_0_TaskPriority_Startup : UDINT
GET
ContextInfoArr_0_TaskPriority_Startup := stInitData.ContextInfoArr_0_TaskPriority;
END_GET
SET
stInitData.ContextInfoArr_0_TaskPriority := ContextInfoArr_0_TaskPriority_Startup;
END_SET
END_PROPERTY

PROPERTY ContextInfoArr_0_TaskSortOrder_Online : UDINT
GET
hResult := GetObjPara(16#030020b0,sizeof(ContextInfoArr_0_TaskSortOrder_Online),adr(ContextInfoArr_0_TaskSortOrder_Online));
END_GET
SET
hResult := SetObjPara(16#030020b0,sizeof(ContextInfoArr_0_TaskSortOrder_Online),adr(ContextInfoArr_0_TaskSortOrder_Online));
END_SET
END_PROPERTY

PROPERTY ContextInfoArr_0_TaskSortOrder_Startup : UDINT
GET
ContextInfoArr_0_TaskSortOrder_Startup := stInitData.ContextInfoArr_0_TaskSortOrder;
END_GET
SET
stInitData.ContextInfoArr_0_TaskSortOrder := ContextInfoArr_0_TaskSortOrder_Startup;
END_SET
END_PROPERTY

PROPERTY CycleUpdateExecuted_Online : BOOL
GET
hResult := GetObjPara(16#00000004,sizeof(CycleUpdateExecuted_Online),adr(CycleUpdateExecuted_Online));
END_GET
SET
hResult := SetObjPara(16#00000004,sizeof(CycleUpdateExecuted_Online),adr(CycleUpdateExecuted_Online));
END_SET
END_PROPERTY

METHOD Execute : HRESULT

IF (SUCCEEDED(hResult)) THEN
  hResult := VerifyParameters();
END_IF

	// update DataArea information
SetDataAreaInfo(ADR(arrDataAreas),2);
	
	// call base method
Execute := SUPER^.Execute();
END_METHOD

PROPERTY ExecuteModelCode_Online : BOOL
GET
hResult := GetObjPara(16#00000008,sizeof(ExecuteModelCode_Online),adr(ExecuteModelCode_Online));
END_GET
SET
hResult := SetObjPara(16#00000008,sizeof(ExecuteModelCode_Online),adr(ExecuteModelCode_Online));
END_SET
END_PROPERTY

PROPERTY ExecuteModelCode_Startup : BOOL
GET
ExecuteModelCode_Startup := stInitData.ExecuteModelCode;
END_GET
SET
stInitData.ExecuteModelCode := ExecuteModelCode_Startup;
END_SET
END_PROPERTY

PROPERTY ExecutionSequence_Online : TctModuleExecutionSequenceType
GET
hResult := GetObjPara(16#00000001,sizeof(ExecutionSequence_Online),adr(ExecutionSequence_Online));
END_GET
SET
hResult := SetObjPara(16#00000001,sizeof(ExecutionSequence_Online),adr(ExecutionSequence_Online));
END_SET
END_PROPERTY

PROPERTY ExecutionSequence_Startup : TctModuleExecutionSequenceType
GET
ExecutionSequence_Startup := stInitData.ExecutionSequence;
END_GET
SET
stInitData.ExecutionSequence := ExecutionSequence_Startup;
END_SET
END_PROPERTY

METHOD FB_init : BOOL
VAR_INPUT
	/// if TRUE, the retain variables are initialized (warm start / cold start)
	bInitRetains: BOOL;
	/// if TRUE, the instance afterwards gets moved into the copy code (online change)
	bInCopyCode: BOOL;
	oid: OTCID;
END_VAR
VAR
	clsId: CLSID;
END_VAR

// initialize flags
bParametersVerified := false;
                    
// set module class id for compatibility check
clsId.Data1 := 16#17344ca2;
clsId.Data2 := 16#8deb;
clsId.Data3 := 16#423e;
clsId.Data4[0] := 16#86;
clsId.Data4[1] := 16#b2;
clsId.Data4[2] := 16#c0;
clsId.Data4[3] := 16#72;
clsId.Data4[4] := 16#d9;
clsId.Data4[5] := 16#0e;
clsId.Data4[6] := 16#c9;
clsId.Data4[7] := 16#86;

AssignClassId(clsId);
                    
// initialize InitData structure with default values              
stInitData.CallByHdr.indexGroup := 0;
stInitData.CallByHdr.indexOffset := 16#00000000;
stInitData.CallByHdr.cbData := SIZEOF(stInitData.CallBy);
stInitData.CallBy := TctModuleCallByType.Module;
stInitData.ExecutionSequenceHdr.indexGroup := 0;
stInitData.ExecutionSequenceHdr.indexOffset := 16#00000001;
stInitData.ExecutionSequenceHdr.cbData := SIZEOF(stInitData.ExecutionSequence);
stInitData.ExecutionSequence := TctModuleExecutionSequenceType.StateUpdateAfterOutputMapping;
stInitData.StepSizeHdr.indexGroup := 0;
stInitData.StepSizeHdr.indexOffset := 16#00000002;
stInitData.StepSizeHdr.cbData := SIZEOF(stInitData.StepSize);
stInitData.StepSize := TctStepSizeType.UseTaskCycleTime;
stInitData.ExecuteModelCodeHdr.indexGroup := 0;
stInitData.ExecuteModelCodeHdr.indexOffset := 16#00000008;
stInitData.ExecuteModelCodeHdr.cbData := SIZEOF(stInitData.ExecuteModelCode);
stInitData.ExecuteModelCode := 1;
stInitData.ContextInfoArr_0_TaskOidHdr.indexGroup := 0;
stInitData.ContextInfoArr_0_TaskOidHdr.indexOffset := 16#03002060;
stInitData.ContextInfoArr_0_TaskOidHdr.cbData := SIZEOF(stInitData.ContextInfoArr_0_TaskOid);
stInitData.ContextInfoArr_0_TaskPriorityHdr.indexGroup := 0;
stInitData.ContextInfoArr_0_TaskPriorityHdr.indexOffset := 16#03002070;
stInitData.ContextInfoArr_0_TaskPriorityHdr.cbData := SIZEOF(stInitData.ContextInfoArr_0_TaskPriority);
stInitData.ContextInfoArr_0_TaskCycleTimeNsHdr.indexGroup := 0;
stInitData.ContextInfoArr_0_TaskCycleTimeNsHdr.indexOffset := 16#03002080;
stInitData.ContextInfoArr_0_TaskCycleTimeNsHdr.cbData := SIZEOF(stInitData.ContextInfoArr_0_TaskCycleTimeNs);
stInitData.ContextInfoArr_0_TaskPortHdr.indexGroup := 0;
stInitData.ContextInfoArr_0_TaskPortHdr.indexOffset := 16#03002090;
stInitData.ContextInfoArr_0_TaskPortHdr.cbData := SIZEOF(stInitData.ContextInfoArr_0_TaskPort);
stInitData.ContextInfoArr_0_TaskSortOrderHdr.indexGroup := 0;
stInitData.ContextInfoArr_0_TaskSortOrderHdr.indexOffset := 16#030020b0;
stInitData.ContextInfoArr_0_TaskSortOrderHdr.cbData := SIZEOF(stInitData.ContextInfoArr_0_TaskSortOrder);
stInitData.Header.cbData := SIZEOF(stInitData)-SIZEOF(stInitData.Header);
stInitData.Header.uiElmCnt := 9;


// set pointer to InitData structure
SetInitDataInfo(ADR(stInitData));

// set DataArea information
SetDataAreaInfo(ADR(arrDataAreas),2);
arrDataAreas[1].nDataAreaId := 0;
arrDataAreas[1].nSize := SIZEOF(stInput);
arrDataAreas[1].pPlcVar := ADR(stInput);
arrDataAreas[1].pModuleProcImg := 0;
arrDataAreas[1].eDataAreaType := E_TcMatSimDataAreaType.InputDst;
arrDataAreas[2].nDataAreaId := 1;
arrDataAreas[2].nSize := SIZEOF(stOutput);
arrDataAreas[2].pPlcVar := ADR(stOutput);
arrDataAreas[2].pModuleProcImg := 0;
arrDataAreas[2].eDataAreaType := E_TcMatSimDataAreaType.OutputSrc;


// initialize basic interface pointers and return
FB_init := SUCCEEDED(Init(oid));
END_METHOD

PROPERTY InitData : ST_HexMove_InitData
GET
InitData := stInitData;
END_GET
SET
stInitData := InitData;
END_SET
END_PROPERTY

PROPERTY Input_Online : ExtU_hexmove_T
GET
hResult := GetObjPara(16#80000000,sizeof(Input_Online),adr(Input_Online));
END_GET
SET
hResult := SetObjPara(16#80000000,sizeof(Input_Online),adr(Input_Online));
END_SET
END_PROPERTY

{attribute 'object_name' := 'Internal_SetObjState'}
METHOD PROTECTED Internal_SetObjState
VAR_INPUT
	hr: REFERENCE TO HRESULT;
	nextState: TCOM_STATE;
END_VAR

// update pointer to InitData structure
SetInitDataInfo(ADR(stInitData));
// call base method
SUPER^.Internal_SetObjState(hr,nextState);
END_METHOD

PROPERTY MdlInitialized_Online : BOOL
GET
hResult := GetObjPara(16#00000003,sizeof(MdlInitialized_Online),adr(MdlInitialized_Online));
END_GET
SET
hResult := SetObjPara(16#00000003,sizeof(MdlInitialized_Online),adr(MdlInitialized_Online));
END_SET
END_PROPERTY

PROPERTY ModuleBuildInfo_Online : TctModuleBuildInfoType
GET
hResult := GetObjPara(16#00000007,sizeof(ModuleBuildInfo_Online),adr(ModuleBuildInfo_Online));
END_GET
SET
hResult := SetObjPara(16#00000007,sizeof(ModuleBuildInfo_Online),adr(ModuleBuildInfo_Online));
END_SET
END_PROPERTY

PROPERTY ModuleInfo_Online : TctModuleInfoType
GET
hResult := GetObjPara(16#00000006,sizeof(ModuleInfo_Online),adr(ModuleInfo_Online));
END_GET
SET
hResult := SetObjPara(16#00000006,sizeof(ModuleInfo_Online),adr(ModuleInfo_Online));
END_SET
END_PROPERTY

{attribute 'object_name' := 'SaveOnlineParametersForInit'}
METHOD SaveOnlineParametersForInit : HRESULT
VAR
	idx: UINT;
	pInitElemHdr: POINTER TO TComInitDataElmHdr;
	pData: PVOID;
	nData: UDINT;
END_VAR
VAR CONSTANT
	nInitDataAlignment: UDINT := 4;
END_VAR

// update pointer to InitData structure
SetInitDataInfo(ADR(stInitData));
// call base method
SaveOnlineParametersForInit := SUPER^.SaveOnlineParametersForInit();
END_METHOD

PROPERTY SimulinkTime_Online : LREAL
GET
hResult := GetObjPara(16#00000005,sizeof(SimulinkTime_Online),adr(SimulinkTime_Online));
END_GET
SET
hResult := SetObjPara(16#00000005,sizeof(SimulinkTime_Online),adr(SimulinkTime_Online));
END_SET
END_PROPERTY

PROPERTY StepSize_Online : TctStepSizeType
GET
hResult := GetObjPara(16#00000002,sizeof(StepSize_Online),adr(StepSize_Online));
END_GET
SET
hResult := SetObjPara(16#00000002,sizeof(StepSize_Online),adr(StepSize_Online));
END_SET
END_PROPERTY

PROPERTY StepSize_Startup : TctStepSizeType
GET
StepSize_Startup := stInitData.StepSize;
END_GET
SET
stInitData.StepSize := StepSize_Startup;
END_SET
END_PROPERTY

{attribute 'object_name' := 'VerifyParameters'}
METHOD PRIVATE VerifyParameters : HRESULT
VAR
	moduleCallByParam: TctModuleCallByType;
END_VAR

IF (bParametersVerified) THEN
  VerifyParameters := Tc2_System.E_HRESULTAdsErr.HRESULT_ADS_NOERROR;
ELSE
  VerifyParameters := GetObjPara(stInitData.CallByHdr.indexOffset,SIZEOF(moduleCallByParam),ADR(moduleCallByParam));
  
  // check the "CallBy" parameter to be set to "Module"
  IF (SUCCEEDED(VerifyParameters) AND (moduleCallByParam <> TctModuleCallByType.Module)) THEN
      VerifyParameters := Tc2_System.E_HRESULTAdsErr.INVALIDPARM;
  END_IF
  
  // set the parameters verified flag
  bParametersVerified := SUCCEEDED(VerifyParameters);
END_IF
END_METHOD

END_FUNCTION_BLOCK

// ---- GlobalTextList.TcGTLO
TEXTLIST GlobalTextList
  145 = ' %.2f'
  165 = ' t_Interval=%.2f'
  167 = ' t_Interval=%.3f'
  169 = ' t_Interval=%.4f'
  168 = ' t_Interval=%.5f'
  143 = '%.2f'
  81 = 'Axis10_Back'
  82 = 'Axis10_Home'
  117 = 'Axis10_Move'
  11 = 'Axis10_Power'
  83 = 'Axis11_Back'
  84 = 'Axis11_Home'
  118 = 'Axis11_Move'
  12 = 'Axis11_Power'
  85 = 'Axis12_Back'
  86 = 'Axis12_Home'
  119 = 'Axis12_Move'
  13 = 'Axis12_Power'
  87 = 'Axis13_Back'
  88 = 'Axis13_Home'
  120 = 'Axis13_Move'
  14 = 'Axis13_Power'
  89 = 'Axis14_Back'
  90 = 'Axis14_Home'
  121 = 'Axis14_Move'
  15 = 'Axis14_Power'
  91 = 'Axis15_Back'
  92 = 'Axis15_Home'
  122 = 'Axis15_Move'
  16 = 'Axis15_Power'
  93 = 'Axis16_Back'
  94 = 'Axis16_Home'
  123 = 'Axis16_Move'
  17 = 'Axis16_Power'
  95 = 'Axis17_Back'
  96 = 'Axis17_Home'
  124 = 'Axis17_Move'
  18 = 'Axis17_Power'
  97 = 'Axis18_Back'
  98 = 'Axis18_Home'
  125 = 'Axis18_Move'
  19 = 'Axis18_Power'
  62 = 'Axis1_Back'
  64 = 'Axis1_Home'
  63 = 'Axis1_Home_Set'
  106 = 'Axis1_M'
  108 = 'Axis1_Move'
  2 = 'Axis1_Power'
  65 = 'Axis2_Back'
  66 = 'Axis2_Home'
  109 = 'Axis2_Move'
  3 = 'Axis2_Power'
  67 = 'Axis3_Back'
  68 = 'Axis3_Home'
  110 = 'Axis3_Move'
  4 = 'Axis3_Power'
  69 = 'Axis4_Back'
  70 = 'Axis4_Home'
  111 = 'Axis4_Move'
  5 = 'Axis4_Power'
  71 = 'Axis5_Back'
  72 = 'Axis5_Home'
  112 = 'Axis5_Move'
  6 = 'Axis5_Power'
  73 = 'Axis6_Back'
  74 = 'Axis6_Home'
  113 = 'Axis6_Move'
  7 = 'Axis6_Power'
  75 = 'Axis7_Back'
  76 = 'Axis7_Home'
  114 = 'Axis7_Move'
  8 = 'Axis7_Power'
  77 = 'Axis8_Back'
  78 = 'Axis8_Home'
  115 = 'Axis8_Move'
  9 = 'Axis8_Power'
  79 = 'Axis9_Back'
  80 = 'Axis9_Home'
  116 = 'Axis9_Move'
  10 = 'Axis9_Power'
  56 = 'Axis_ActPostion[INDEX]'
  60 = 'Back'
  57 = 'Current_Turque_Value[INDEX]'
  39 = 'Driver10_Reset'
  40 = 'Driver11_Reset'
  41 = 'Driver12_Reset'
  42 = 'Driver13_Reset'
  43 = 'Driver14_Reset'
  44 = 'Driver15_Reset'
  45 = 'Driver16_Reset'
  46 = 'Driver17_Reset'
  47 = 'Driver18_Reset'
  30 = 'Driver1_Reset'
  31 = 'Driver2_Reset'
  32 = 'Driver3_Reset'
  33 = 'Driver4_Reset'
  34 = 'Driver5_Reset'
  35 = 'Driver6_Reset'
  36 = 'Driver7_Reset'
  37 = 'Driver8_Reset'
  38 = 'Driver9_Reset'
  127 = 'Error & Reset'
  126 = 'Error&Reset'
  151 = 'Exsetopint_Enable'
  152 = 'Exsetopint_On'
  141 = 'Exsetpoint_Exectue'
  23 = 'Home'
  59 = 'Home_Execute'
  61 = 'Home_Set'
  131 = 'Leg1_Home'
  132 = 'Leg2_Home'
  133 = 'Leg3_Home'
  134 = 'Leg4_Home'
  135 = 'Leg5_Home'
  136 = 'Leg6_Home'
  130 = 'Move & Stand'
  107 = 'MoveAbsoluteDone[INDEX]'
  129 = 'Move_Execute'
  53 = 'Power'
  20 = 'Power_Execute'
  29 = 'Reset'
  49 = 'Reset_Execute'
  26 = 'Robot_Error'
  101 = 'Robot_Home_Set'
  0 = 'Robot_Power'
  48 = 'Robot_Reset'
  128 = 'Robot_Stand_Execute'
  99 = 'Robot_Start_Back'
  100 = 'sadad'
  166 = 'Simulink_Move'
  147 = 't=%.2f'
  170 = 't=%.3f'
  144 = 'T_ALL = %.2f'
  158 = 't_Interval=%.2f'
  22 = '切换视图'
  157 = '取样时间间隔 t_Interval'
  160 = '取样时间间隔 t_Interval(ms)'
  161 = '取样时间间隔 t_Interval(s)'
  159 = '取样时间间隔 t_Interval/ms'
  139 = '可以用来整体机器人运动'
  140 = '可以用来整体机器人进行Simulink模型验证'
  104 = '可以用来给单个四缸伸长或者是整体机器人站立'
  28 = '可以用来给单个电机或者是整体机器人上电'
  55 = '可以用来给单个电机或者是整体机器人找零'
  103 = '可以用来给单个电机或者是整体机器人站立'
  52 = '可以用来错误时给单个电机或者是整体机器人进行驱动重置'
  24 = '否'
  149 = '开始输入轨迹'
  156 = '当前取样时间 t'
  163 = '当前取样时间 t(s)'
  25 = '是'
  148 = '是否开始输入轨迹'
  21 = '是否进行上电操作'
  58 = '是否进行找零操作'
  1 = '是否进行整机操作'
  142 = '是否进行运动操作'
  50 = '是否进行驱动重置'
  138 = '本界面为电机Sumulink模型运动程序：'
  137 = '本界面为电机Sumulink程序：'
  27 = '本界面为电机上电程序：'
  102 = '本界面为电机伸长/机器人站立程序：'
  54 = '本界面为电机找零程序：'
  105 = '本界面为电机绝对运动/机器人站立程序：'
  51 = '本界面为驱动重置程序：'
  154 = '输入运动总时长 T_ALL'
  162 = '输入运动总时长 T_ALL(s)'
  150 = '运动当前时间 t'
  164 = '运动当前时间 t(s)'
  146 = '运动总时长 T_ALL'
  155 = '运动时间间隔 t'
  153 = '运动终止信号'
END_TEXTLIST

// ---- VISUs/Visu_SimulinkMove.TcVIS
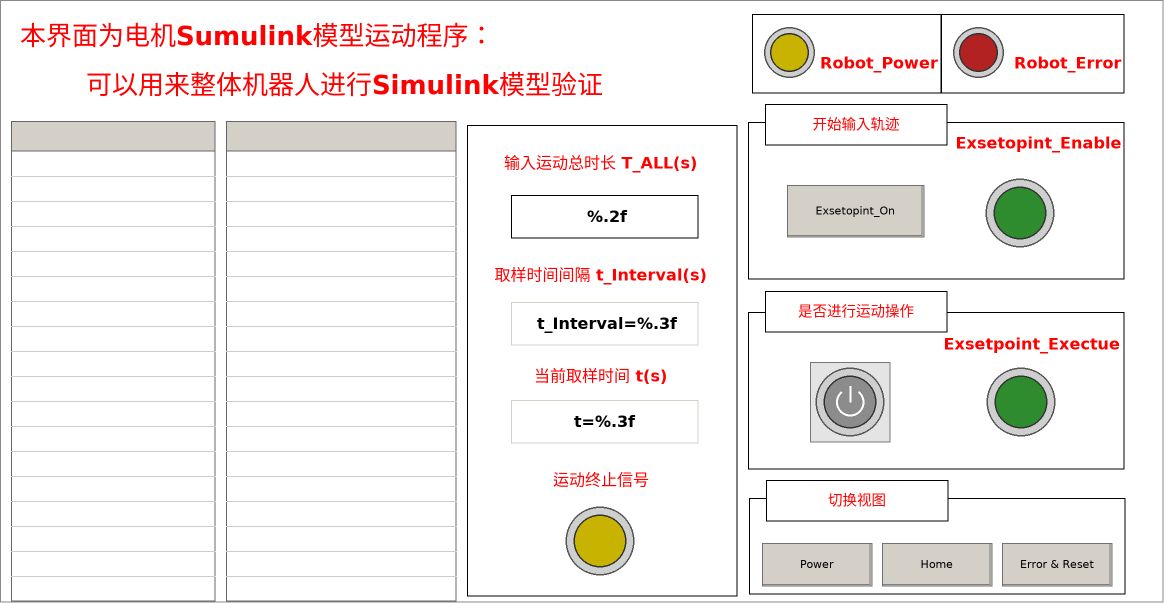
VISUALIZATION Visu_SimulinkMove  // 1164x603
    Rectangle (749,498 376x96)
    Rectangle (766,480 182x41), "切换视图"
    Button (762,543 110x43), "Power"
        OnMouseClick: change screen: Visu_Power
    Button (1002,543 110x43), "Error & Reset"
        OnMouseClick: change screen: Visu_Reset
    Button (882,543 110x43), "Home"
        OnMouseClick: change screen: Visu_Home
    Rectangle (467,125 270x471)
    Rectangle (752,14 189x79)
    Rectangle (748,312 376x157)
    Label (902,328 260x32), "Exsetpoint_Exectue"
    Rectangle (765,291 182x41), "是否进行运动操作"
    Lamp1 (981,362 80x80), variable: MAIN.ExSetPoint_Execute, style: Lamp-Lamp1-Green
    PowerSwitch (810,362 80x80), variable: MAIN.ExSetPoint_Execute, behaviour: TOGGLE, style: Switch-PowerSwitch-Gray
    Rectangle (941,14 183x79)
    Lamp1 (948,23 61x59), variable: MAIN.Robot_Error, style: Lamp-Lamp1-Red
    Label (991,47 154x32), "Robot_Error"
    Label (17,15 572x42), "本界面为电机Sumulink模型运动程序："
    Label (83,64 874x42), "可以用来整体机器人进行Simulink模型验证"
    Table (11,121 204x480), data array: MAIN.Axis_ActPostion
        p3854506369: MAIN.Axis_ActPostion[INDEX]
    Table (226,121 230x480), data array: MAIN.Current_Turque_Value
        p3854506369: MAIN.Current_Turque_Value[INDEX]
    Lamp1 (759,23 61x59), variable: MAIN.Robot_Power, style: Lamp-Lamp1-Yellow
    Label (802,47 154x32), "Robot_Power"
    Rectangle (748,122 376x157)
    Rectangle (765,104 182x41), "开始输入轨迹"
    Lamp1 (980,173 80x80), variable: MAIN.ExtSetPointEnable, style: Lamp-Lamp1-Green
    Label (935,127 207x32), "Exsetopint_Enable"
    Rectangle (511,195 187x43), "%.2f", text variable: MAIN.T_All
        OnMouseClick: write MAIN.T_All via Default
    Label (471,147 260x32), "输入运动总时长 T_ALL(s)"
    Textfield (511,400 187x43), "t=%.3f", text variable: MAIN.t
    Label (471,360 260x32), "当前取样时间 t(s)"
    Button (787,185 137x52), "Exsetopint_On"
        toggle MAIN.ExtSetPointEnable
    Lamp1 (560,501 80x80), variable: MAIN.ExtSetPointDisable, style: Lamp-Lamp1-Yellow
    Label (471,464 260x32), "运动终止信号"
    Label (471,259 260x32), "取样时间间隔 t_Interval(s)"
    Textfield (511,302 187x43), "t_Interval=%.3f", text variable: MAIN.t_Interval
        OnMouseClick: write MAIN.t_Interval via Default
END_VISUALIZATION
